# EPICS autosave request: MDrive/MDriveSettings.req
# Motor record settings
# Real motors
file "motor_settings.req" P=$(P), M=m1
file "motor_settings.req" P=$(P), M=m2
file "motor_settings.req" P=$(P), M=m3
file "motor_settings.req" P=$(P), M=m4
